// Mitsubishi GX Works2 project: 16-06-2020 TA1_Ex4   PLC: FX3G

PROGRAM MAIN
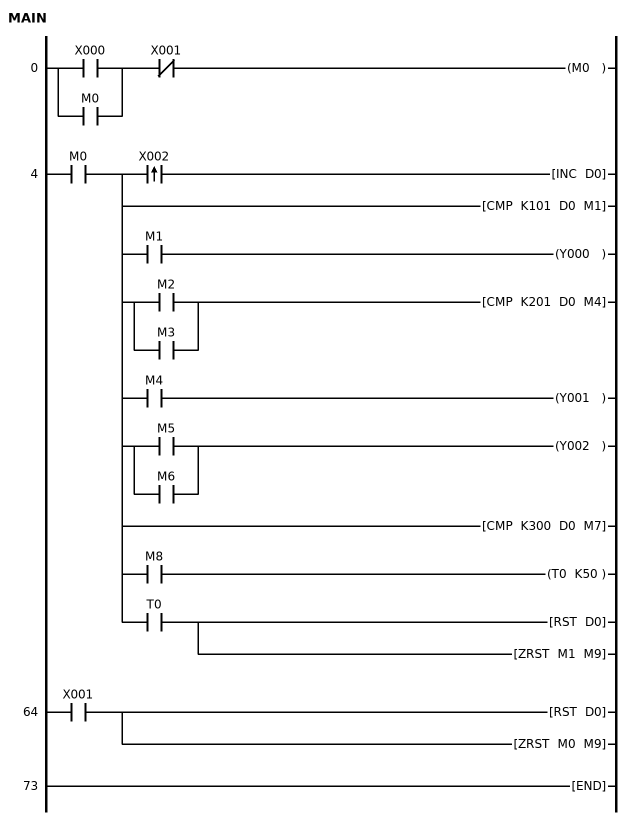
0     LD      X000
      OR      M0
      ANI     X001
      OUT     M0
4     LD      M0
      MPS
      ANDP    X002
      INC     D0
      MPP
      CMP     K101 D0 M1
      MPS
      AND     M1
      OUT     Y000
      MRD
      LD      M2
      OR      M3
      ANB
      CMP     K201 D0 M4
      MRD
      AND     M4
      OUT     Y001
      MRD
      LD      M5
      OR      M6
      ANB
      OUT     Y002
      MPP
      CMP     K300 D0 M7
      MPS
      AND     M8
      OUT     T0 K50
      MPP
      AND     T0
      RST     D0
      ZRST    M1 M9
64    LD      X001
      RST     D0
      ZRST    M0 M9
73    END
END_PROGRAM
